(* 
    This testsuite verifies that the Assert_True and Assert_False methods do what they are supposed to. It does so
    by making sure that every assert-method (assert_true & assert_false) does both one failing and one successful
    assert.
*)
FUNCTION_BLOCK FB_AssertTrueFalse EXTENDS TcUnit.FB_TestSuite

AssertThatINTsAreEqual();
AssertThatINTsAreNotEqual();
AssertThatWORDsAreEqual();
AssertThatWORDsAreNotEqual();

METHOD PRIVATE AssertThatINTsAreEqual
VAR
    a : INT := -33;
    b : INT := -44;
END_VAR
TEST('AssertThatINTsAreEqual');

AssertFalse(Condition := (a <> b),
            Message := 'INTs are equal');

TEST_FINISHED();
END_METHOD

METHOD PRIVATE AssertThatINTsAreNotEqual
VAR
    a : INT := -33;
    b : INT := -44;
END_VAR
TEST('AssertThatINTsAreNotEqual');

AssertFalse(Condition := (a = b),
            Message := 'INTs are equal');

TEST_FINISHED();
END_METHOD

METHOD PRIVATE AssertThatWORDsAreEqual
VAR
    a : WORD := 16#ABCD;
    b : WORD := 16#0123;
END_VAR
TEST('AssertThatWORDsAreEqual');

AssertTrue(Condition := (a = b),
           Message := 'WORDs are not equal');

TEST_FINISHED();
END_METHOD

METHOD PRIVATE AssertThatWORDsAreNotEqual
VAR
    a : WORD := 16#ABCD;
    b : WORD := 16#0123;
END_VAR
TEST('AssertThatWORDsAreNotEqual');

AssertTrue(Condition := (a <> b),
           Message := 'WORDs are equal');

TEST_FINISHED();
END_METHOD

END_FUNCTION_BLOCK

(* stored: Version 1.1.0.1, ProductVersion 3.1.4022.18
   POU FB_AssertTrueFalse: Id {4a344c15-007d-4e24-b34e-25e793163fe6}, SpecialFunc None
   Method AssertThatINTsAreEqual: Id {e329edff-158b-47b8-b448-4482e312fc51}
   Method AssertThatINTsAreNotEqual: Id {e9713416-6687-4536-b3eb-d0e312881039}
   Method AssertThatWORDsAreEqual: Id {cb8a8728-6b7f-485b-9255-e9e2c3d7b1b4}
   Method AssertThatWORDsAreNotEqual: Id {7f2e9dc0-aaa1-4524-9220-4e31b7d76d84} *)
